// TIA Portal V17 export
// export: Created 2023-02-25T15:48:37.1830141Z, ExportSetting WithDefaults, DisplayName Totally Integrated Automation Portal, DisplayVersion V17, DisplayName TIA Portal Openness, DisplayVersion V17, DisplayName TIA Portal Version Control Interface, DisplayVersion V17, DisplayName TIA Portal Test Suite Advanced, DisplayVersion V17, DisplayName STEP 7 Professional, DisplayVersion V17, DisplayName SIMATIC Energy Suite, DisplayVersion V17, DisplayName STEP 7 Safety, DisplayVersion V17, DisplayName WinCC Professional, DisplayVersion V17
TYPE "stt_Conveyor"
// stored: IsFailsafeCompliant false
   STRUCT
      C1 : Bool;
      C2 { S7_SetPoint := 'True'} : Bool;
      C3 { S7_SetPoint := 'True'} : Bool;
      C4 { S7_SetPoint := 'True'} : Bool;
      W { S7_SetPoint := 'True'} : Bool;
      Left : Bool;
      Forward : Bool;
      Right : Bool;
   END_STRUCT;
END_TYPE
